// TIA Portal V21 export
TYPE "Std_RitSoglia"
   STRUCT
      Maxi : "Std_stTimer";
      IntMax { S7_SetPoint := 'True'} : "Std_stTimer";
      IntMin { S7_SetPoint := 'True'} : "Std_stTimer";
      Mini { S7_SetPoint := 'True'} : "Std_stTimer";
   END_STRUCT;
END_TYPE
